{attribute addProperty BoxType "EK1122-0000-0018"}
{attribute addProperty Id "Beckhoff_EL69xxsub_EK1100EK1100_179A0949162"}
{attribute addProperty CRC "2729636568"}
{attribute addProperty SizeInBites "16"}
{attribute addProperty SizeInBytes "2"}
TYPE Beckhoff_EL69xxEK1122_A2B2F2D8 EXTENDS EK1122_179A0949 :
STRUCT
	{attribute addProperty Name "Beckhoff_EL69xxsub_EK1100"}
	Beckhoff_EL69xxsub_EK1100 : EK1100_179A0949;
END_STRUCT
END_TYPE

(* stored: Version 1.2.0.0, ProductVersion 3.1.4024.9
   DUT Beckhoff_EL69xxEK1122_A2B2F2D8: Id {ccb3a55c-6e50-4c15-9289-5066628527a9} *)
